// TIA Portal V15.1 export
// export: Created 2024-06-21T08:40:41.4904848Z, ExportSetting WithDefaults, DisplayName Totally Integrated Automation Portal, DisplayVersion V15.1 Update 5, DisplayName TIA Portal Openness, DisplayVersion V15.1 Update 5, DisplayName SINAMICS Startdrive Advanced, DisplayVersion V15.1, DisplayName G130, G150, S120, S150, SINAMICS MV, S210, DisplayVersion V15.1, DisplayName G110M, G120, G120C, G120D, G120P, DisplayVersion V15.1, DisplayName STEP 7 Professional, DisplayVersion V15.1 Update 5, DisplayName STEP 7 Safety, DisplayVersion V15.1, DisplayName WinCC Professional, DisplayVersion V15.1 Update 5, DisplayName SIMATIC Visualization Architect, DisplayVersion V15.1
DATA_BLOCK "_PNComPLC308"   // DB260
{ S7_Optimized_Access := 'FALSE' }
AUTHOR : VCG
FAMILY : LocFncGn
NAME : 2011Intf
VERSION : 0.1
// stored: AutoNumber false, DBAccessibleFromOPCUA true, IsOnlyStoredInLoadMemory false, IsWriteProtectedInAS false
   VAR RETAIN
      AA_FPNComAlarm { ExternalAccessible := 'False'; ExternalVisible := 'False'; ExternalWritable := 'False'} : Bool;   // Alarm PN communication with PLC308 (Safety) / Alarm PN communication with PLCyyy (Safety)
      AA_PNComCheckAlarm { ExternalAccessible := 'False'; ExternalVisible := 'False'; ExternalWritable := 'False'} : Bool;   // Alarm PN communication with PLC308 (LiveBit) / Alarm PN communication with PLCyyy (LiveBit)
      PLC308LPNCheckAlarmABCondition { ExternalAccessible := 'False'; ExternalVisible := 'False'; ExternalWritable := 'False'} : Bool;   // Alarm AB condition
      PLC308LPNDiagAlarmABCondition { ExternalAccessible := 'False'; ExternalVisible := 'False'; ExternalWritable := 'False'} : Bool;   // Alarm AB condition
      H_InBit0_15Anim : Word;   // Animation word for HMI
      H_TxtInBit0_15Anim : Struct   // Animation description of the bits
         "0" : String[50];   // Description
         "1" : String[50];   // Description
         "2" : String[50];   // Description
         "3" : String[50];   // Description
         "4" : String[50];   // Description
         "5" : String[50];   // Description
         "6" : String[50];   // Description
         "7" : String[50];   // Description
         "8" : String[50];   // Description
         "9" : String[50];   // Description
         "10" : String[50];   // Description
         "11" : String[50];   // Description
         "12" : String[50];   // Description
         "13" : String[50];   // Description
         "14" : String[50];   // Description
         "15" : String[50];   // Description
      END_STRUCT;
      H_InBit16_31Anim : Word;   // Animation word for HMI
      H_TxtInBit16_31Anim : Struct   // Animation description of the bits
         "0" : String[50];   // Description
         "1" : String[50];   // Description
         "2" : String[50];   // Description
         "3" : String[50];   // Description
         "4" : String[50];   // Description
         "5" : String[50];   // Description
         "6" : String[50];   // Description
         "7" : String[50];   // Description
         "8" : String[50];   // Description
         "9" : String[50];   // Description
         "10" : String[50];   // Description
         "11" : String[50];   // Description
         "12" : String[50];   // Description
         "13" : String[50];   // Description
         "14" : String[50];   // Description
         "15" : String[50];   // Description
      END_STRUCT;
      H_OutBit0_15Anim : Word;   // Animation word for HMI
      H_TxtOutBit0_15Anim : Struct   // Animation description of the bits
         "0" : String[50];   // Description
         "1" : String[50];   // Description
         "2" : String[50];   // Description
         "3" : String[50];   // Description
         "4" : String[50];   // Description
         "5" : String[50];   // Description
         "6" : String[50];   // Description
         "7" : String[50];   // Description
         "8" : String[50];   // Description
         "9" : String[50];   // Description
         "10" : String[50];   // Description
         "11" : String[50];   // Description
         "12" : String[50];   // Description
         "13" : String[50];   // Description
         "14" : String[50];   // Description
         "15" : String[50];   // Description
      END_STRUCT;
      H_OutBit16_31Anim : Word;   // Animation word for HMI
      H_TxtOutBit16_31Anim : Struct   // Animation description of the bits
         "0" : String[50];   // Description
         "1" : String[50];   // Description
         "2" : String[50];   // Description
         "3" : String[50];   // Description
         "4" : String[50];   // Description
         "5" : String[50];   // Description
         "6" : String[50];   // Description
         "7" : String[50];   // Description
         "8" : String[50];   // Description
         "9" : String[50];   // Description
         "10" : String[50];   // Description
         "11" : String[50];   // Description
         "12" : String[50];   // Description
         "13" : String[50];   // Description
         "14" : String[50];   // Description
         "15" : String[50];   // Description
      END_STRUCT;
      H_FInBit0_15Anim : Word;   // Animation word for HMI
      H_TxtFInBit0_15Anim : Struct   // Animation description of the bits
         "0" : String[50];   // Description
         "1" : String[50];   // Description
         "2" : String[50];   // Description
         "3" : String[50];   // Description
         "4" : String[50];   // Description
         "5" : String[50];   // Description
         "6" : String[50];   // Description
         "7" : String[50];   // Description
         "8" : String[50];   // Description
         "9" : String[50];   // Description
         "10" : String[50];   // Description
         "11" : String[50];   // Description
         "12" : String[50];   // Description
         "13" : String[50];   // Description
         "14" : String[50];   // Description
         "15" : String[50];   // Description
      END_STRUCT;
      H_FOutBit0_15Anim : Word;   // Animation word for HMI
      H_TxtFOutBit0_15Anim : Struct   // Animation description of the bits
         "0" : String[50];   // Description
         "1" : String[50];   // Description
         "2" : String[50];   // Description
         "3" : String[50];   // Description
         "4" : String[50];   // Description
         "5" : String[50];   // Description
         "6" : String[50];   // Description
         "7" : String[50];   // Description
         "8" : String[50];   // Description
         "9" : String[50];   // Description
         "10" : String[50];   // Description
         "11" : String[50];   // Description
         "12" : String[50];   // Description
         "13" : String[50];   // Description
         "14" : String[50];   // Description
         "15" : String[50];   // Description
      END_STRUCT;
      H_PLC308LPNDiagIAnim : Word;   // Animation word for HMI
      H_PLC308LPNCheckIAnim : Word;   // Animation word for HMI
      H_Anim : Word;   // Animation
      H_DBnr : Int;   // DB number
      H_HMICmd : Word;   // HMI command
      H_209230NCB01_Routing : Int;   // Animation Routing Information
      AlarmA { ExternalAccessible := 'False'; ExternalVisible := 'False'; ExternalWritable := 'False'} : Bool;   // Alarm A
      AlarmB { ExternalAccessible := 'False'; ExternalVisible := 'False'; ExternalWritable := 'False'} : Bool;   // Alarm B
      AlarmC { ExternalAccessible := 'False'; ExternalVisible := 'False'; ExternalWritable := 'False'} : Bool;   // Alarm C
      AlarmD { ExternalAccessible := 'False'; ExternalVisible := 'False'; ExternalWritable := 'False'} : Bool;   // Alarm D
      AlarmABCondition { ExternalAccessible := 'False'; ExternalVisible := 'False'; ExternalWritable := 'False'} : Bool;   // Alarm AB condition
      "______308240CR27 --> 210CR21______" { ExternalAccessible := 'False'; ExternalVisible := 'False'; ExternalWritable := 'False'} : Bool;   // -----------------------------------------------------------------------------------
      "308230ZS01AccessStopRequest" { ExternalAccessible := 'False'; ExternalVisible := 'False'; ExternalWritable := 'False'} : Bool;   // Access Stop Request
      "308240AS30ResetPB" { ExternalAccessible := 'False'; ExternalVisible := 'False'; ExternalWritable := 'False'} : Bool;   // AS Light Curtain - Push button Reset
      "308240AS30StartPB" { ExternalAccessible := 'False'; ExternalVisible := 'False'; ExternalWritable := 'False'} : Bool;   // AS Light Curtain - Push button Start
      "308240AS30StopPB" { ExternalAccessible := 'False'; ExternalVisible := 'False'; ExternalWritable := 'False'} : Bool;   // AS Light Curtain - Push button Stop
      "308240ZM01IAnim" { ExternalAccessible := 'False'; ExternalVisible := 'False'; ExternalWritable := 'False'} : Word;   // For animation of icon
      "308240ZM01Modes" { ExternalAccessible := 'False'; ExternalVisible := 'False'; ExternalWritable := 'False'} : "Modes";   // Modes
      "308240CR27" { ExternalAccessible := 'False'; ExternalVisible := 'False'; ExternalWritable := 'False'} : "Conveyor";   // Transfer
      "______308220CR28 --> 220CR21______" { ExternalAccessible := 'False'; ExternalVisible := 'False'; ExternalWritable := 'False'} : Bool;   // -----------------------------------------------------------------------------------
      "308210ZS01AccessStopRequest" { ExternalAccessible := 'False'; ExternalVisible := 'False'; ExternalWritable := 'False'} : Bool;   // Access Stop Request
      "308220AS30ResetPB" { ExternalAccessible := 'False'; ExternalVisible := 'False'; ExternalWritable := 'False'} : Bool;   // AS Light Curtain - Push button Reset
      "308220AS30StartPB" { ExternalAccessible := 'False'; ExternalVisible := 'False'; ExternalWritable := 'False'} : Bool;   // AS Light Curtain - Push button Start
      "308220AS30StopPB" { ExternalAccessible := 'False'; ExternalVisible := 'False'; ExternalWritable := 'False'} : Bool;   // AS Light Curtain - Push button Stop
      "308220ZM01IAnim" { ExternalAccessible := 'False'; ExternalVisible := 'False'; ExternalWritable := 'False'} : Word;   // For animation of icon
      "308210ZM01Modes" { ExternalAccessible := 'False'; ExternalVisible := 'False'; ExternalWritable := 'False'} : "Modes";   // Modes
      "308220ZM01Modes" { ExternalAccessible := 'False'; ExternalVisible := 'False'; ExternalWritable := 'False'} : "Modes";   // Modes
      "308220CR28" { ExternalAccessible := 'False'; ExternalVisible := 'False'; ExternalWritable := 'False'} : "Conveyor";   // Transfer
      "______308220CR25 --> 230CR22______" { ExternalAccessible := 'False'; ExternalVisible := 'False'; ExternalWritable := 'False'} : Bool;   // -----------------------------------------------------------------------------------
      "308210ZS01SafetyOk" { ExternalAccessible := 'False'; ExternalVisible := 'False'; ExternalWritable := 'False'} : Bool;   // Safety Ok
      "308210ZS01PowerOnRequest" { ExternalAccessible := 'False'; ExternalVisible := 'False'; ExternalWritable := 'False'} : Bool;   // Power On Request
      "308210ZS01ResetSafety" { ExternalAccessible := 'False'; ExternalVisible := 'False'; ExternalWritable := 'False'} : Bool;   // Reset Safety
      "308220CR25" { ExternalAccessible := 'False'; ExternalVisible := 'False'; ExternalWritable := 'False'} : "Conveyor";   // Transfer
   END_VAR
BEGIN
END_DATA_BLOCK
